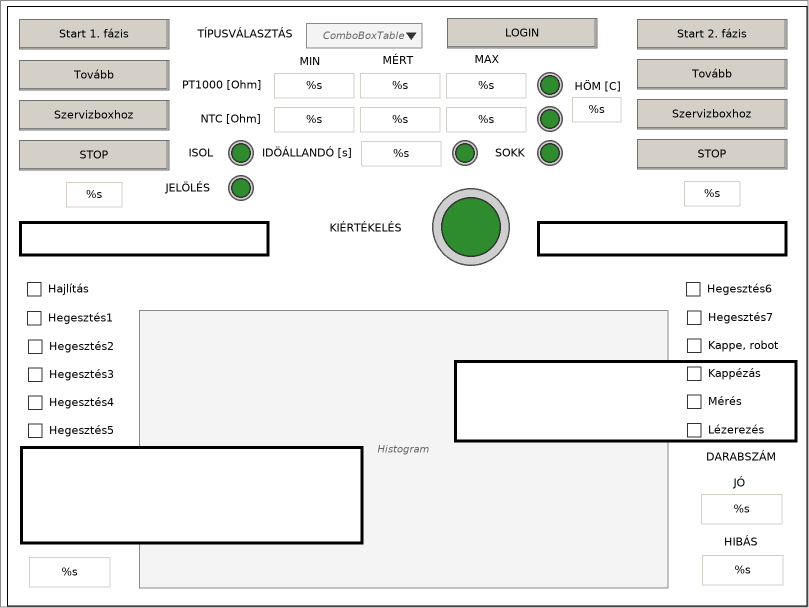
VISUALIZATION Termeles  // 809x608
    Rectangle (7,6 800x600)
    Group (19,19 150x151)
        Button (0,0 150x30), "Start 1. fázis", input disabled if: AUTOMATA.bStart1GombTiltva
            OnMouseUp: execute { AUTOMATA.iState:=1; }
        Button (0,41 150x30), "Tovább"
            OnMouseUp: execute { AUTOMATA.bContinue:=TRUE; }
        Button (0,121 150x30), "STOP"
            OnMouseUp: execute {
                AUTOMATA.bContinue:=FALSE;
                AUTOMATA.iState:=0;
                AUTOMATA.bWelderReservedBy1:=FALSE;
                AUTOMATA.bRobotReservedBy1:=FALSE;
            }
        Button (0,81 150x30), "Szervizboxhoz"
            OnMouseUp: execute { AUTOMATA.iState:=100; }
    Button (637,19 150x30), "Start 2. fázis", input disabled if: AUTOMATA.bStart2GombTiltva
        OnMouseUp: execute { AUTOMATA.iState2:=1; }
    Button (637,59 150x30), "Tovább"
        OnMouseUp: execute { AUTOMATA.bContinue2:=TRUE; }
    Button (637,99 150x30), "Szervizboxhoz"
        OnMouseUp: execute { AUTOMATA.iState2:=100; }
    Button (637,139 150x30), "STOP"
        OnMouseUp: execute {
            AUTOMATA.bContinue2:=FALSE;
            AUTOMATA.iState2:=0;
            AUTOMATA.bWelderReservedBy2:=FALSE;
            AUTOMATA.bRobotReservedBy2:=FALSE;
            GVL.bAdapterLefogo:=FALSE;
        }
    Group (184,138 72x30)
        Lamp1 (42,0 30x30), variable: GVL.bIsolOK, style: Lamp-Lamp1-Green
        Label (0,5 34x20), "ISOL"
    Label (290,49 40x25), "MIN"
    Histogram (139,310 529x278), scale format: %.1f, scale 0..300
        p1518820177: VEGMERO.arIdoallandoPTTEMP
        p102497268: VEGMERO.arIdoallandoPTTEMP
        p788070771: ARRAY [0..600] OF REAL
    Group (489,138 76x30)
        Lamp1 (46,0 30x30), variable: GVL.bShockOK, style: Lamp-Lamp1-Green
        Label (0,5 42x20), "SOKK"
    Textfield (29,557 81x30), "%s", text variable: GVL.nProductCount1, input disabled if: TRUE
    Label (24,521 82x30), "DARABSZÁM"
    Textfield (701,494 81x30), "%s", text variable: GVL.nGoodProductCount, input disabled if: TRUE
    Label (727,468 25x30), "JÓ"
    Textfield (702,555 81x30), "%s", text variable: GVL.nBadProductCount, input disabled if: TRUE
    Label (720,527 42x30), "HIBÁS"
    Label (700,442 82x30), "DARABSZÁM"
    ComboBoxTable (306,23 116x25), variable: GVL.iSelectedProductType, data array: GVL.saProductTypes
        p3854506369: GVL.saProductTypes[INDEX]
    Label (190,19 110x30), "TÍPUSVÁLASZTÁS"
    Group (25,274 106x171)
        Checkbox (0,0 105x30), "Hajlítás", variable: GVL.bHajlitasBe, input disabled if: AUTOMATA.bFolyamatBeallitas1Tiltva
        Checkbox (0,29 105x30), "Hegesztés1", variable: GVL.bHegesztes1Be, input disabled if: AUTOMATA.bFolyamatBeallitas1Tiltva
        Checkbox (1,58 105x29), "Hegesztés2", variable: GVL.bHegesztes2Be, input disabled if: AUTOMATA.bFolyamatBeallitas1Tiltva
        Checkbox (1,86 105x29), "Hegesztés3", variable: GVL.bHegesztes3Be, input disabled if: AUTOMATA.bFolyamatBeallitas1Tiltva
        Checkbox (1,114 105x29), "Hegesztés4", variable: GVL.bHegesztes4Be, input disabled if: AUTOMATA.bFolyamatBeallitas1Tiltva
        Checkbox (1,142 105x29), "Hegesztés5", variable: GVL.bHegesztes5Be, input disabled if: AUTOMATA.bFolyamatBeallitas1Tiltva
    Group (155,173 101x30)
        Label (0,5 66x20), "JELÖLÉS"
        Lamp1 (71,0 30x30), variable: GVL.bMarkingOK, style: Lamp-Lamp1-Green
    Lamp1 (426,182 90x90), variable: GVL.bProductNOK, style: Lamp-Lamp1-Red
    Lamp1 (426,182 90x90), variable: GVL.bProductOK, invisible if: GVL.bProductNOK, style: Lamp-Lamp1-Green
    Label (320,213 91x30), "KIÉRTÉKELÉS"
    Button (447,18 150x30), "LOGIN"
        OnMouseClick: VisuUserMgmt Type=Login
    RoundedRectangle (20,446 343x98), invisible if: GVL.bHibauzenetNTCRejtve, text list: 'ErrorList1', text index: AUTOMATA.iState
    RoundedRectangle (454,360 343x82), invisible if: GVL.bHibauzenetPtRejtve, text list: 'ErrorList2', text index: AUTOMATA.iState2
    Group (684,274 106x171)
        Checkbox (1,141 105x30), "Lézerezés", variable: GVL.bJelolesBe, input disabled if: AUTOMATA.bFolyamatBeallitas2Tiltva
        Checkbox (0,0 105x30), "Hegesztés6", variable: GVL.bHegesztes6Be, input disabled if: AUTOMATA.bFolyamatBeallitas2Tiltva
        Checkbox (1,29 105x29), "Hegesztés7", variable: GVL.bHegesztes7Be, input disabled if: AUTOMATA.bFolyamatBeallitas2Tiltva
        Checkbox (1,57 105x29), "Kappe, robot", variable: GVL.bRobotKappeBe, input disabled if: AUTOMATA.bFolyamatBeallitas2Tiltva
        Checkbox (1,85 105x29), "Kappézás", variable: GVL.bKappeBe, input disabled if: AUTOMATA.bFolyamatBeallitas2Tiltva
        Checkbox (1,113 105x29), "Mérés", variable: GVL.bMeresBe, input disabled if: AUTOMATA.bFolyamatBeallitas2Tiltva
    RoundedRectangle (19,221 250x35), text list: 'AUTOMATA_lepesek1', text index: AUTOMATA.iState
    RoundedRectangle (537,221 250x35), text list: 'AUTOMATA_lepesek2', text index: AUTOMATA.iState2
    Group (178,70 387x30)
        Label (0,5 88x20), "PT1000 [Ohm]"
        Lamp1 (357,0 30x30), variable: GVL.bPTResOK, style: Lamp-Lamp1-Green
        Textfield (182,3 80x25), "%s", text variable: GVL.rPtRes, input disabled if: TRUE
        Textfield (96,3 80x25), "%s", text variable: VEGMERO.PTRES_MIN, input disabled if: TRUE
        Textfield (268,3 80x25), "%s", text variable: VEGMERO.PTRES_MAX, input disabled if: TRUE
    Label (196,109 70x20), "NTC [Ohm]"
    Lamp1 (535,104 30x30), variable: GVL.bNTCResOK, style: Lamp-Lamp1-Green
    Textfield (360,107 80x25), "%s", text variable: GVL.rPtRes, input disabled if: TRUE
    Textfield (274,107 80x25), "%s", text variable: VEGMERO.NTCRES_MIN, input disabled if: TRUE
    Textfield (446,107 80x25), "%s", text variable: VEGMERO.NTCRES_MAX, input disabled if: TRUE
    Group (256,138 224x30)
        Lamp1 (194,0 30x30), variable: GVL.bTimeConstOK, style: Lamp-Lamp1-Green
        Label (0,5 102x20), "IDÖÁLLANDÓ [s]"
        Textfield (105,3 80x25), "%s", text variable: GVL.rTimeConst, input disabled if: TRUE
    Textfield (572,97 49x25), "%s", text variable: GVL.rTemp, input disabled if: TRUE
    Textfield (66,182 56x25), "%s", text variable: AUTOMATA.iState, input disabled if: TRUE
    Textfield (684,181 56x25), "%s", text variable: AUTOMATA.iState2, input disabled if: TRUE
    Label (467,47 40x25), "MAX"
    Label (378,48 40x25), "MÉRT"
    Label (573,74 50x25), "HÖM [C]"
END_VISUALIZATION

(* stored: Version 1.1.0.1, ProductVersion 3.1.4024.11
   Visu Termeles: Id {708d0646-aebf-4c45-b358-2304fb1aae90} *)
